// Interlock logic for the Baseplate Chiller
FUNCTION F_BaseplateChillerEnable : BOOL
VAR_INPUT
    bMasterOverride : BOOL; //Master manual override control input
END_VAR
VAR_IN_OUT CONSTANT
    stErrors : ST_ErrorStates; // Currently detected errors
END_VAR
VAR
END_VAR

IF (stErrors.bHardwareFailure // Disable baseplate chiller if there is a hardware failure
    (* OR stErrors.bLeakUnderTable *) OR stErrors.bLeakOpcpaCarbideOn) // Disable baseplate chiller if there is a leak under the table
    AND NOT bMasterOverride //if master override is TRUE, ignore all errors
THEN
    F_BaseplateChillerEnable := FALSE;
ELSE
    F_BaseplateChillerEnable := TRUE;
END_IF

END_FUNCTION

(* stored: Version 1.1.0.1, ProductVersion 3.1.4024.6
   POU F_BaseplateChillerEnable: Id {e65513cd-e37f-4070-bd0b-50d5fee18685}, SpecialFunc None *)
